FUNCTION alg_a_zdown : BOOL
VAR_INPUT
	state: STATE;
END_VAR

alg_a_zdown := state.dvar_M_example_controller_a_zdown;

END_FUNCTION

(* stored: Version 1.1.0.1, ProductVersion 3.1.4022.18
   POU alg_a_zdown: Id {48045020-26dc-48b8-996a-5668c0416ea8}, SpecialFunc None *)
